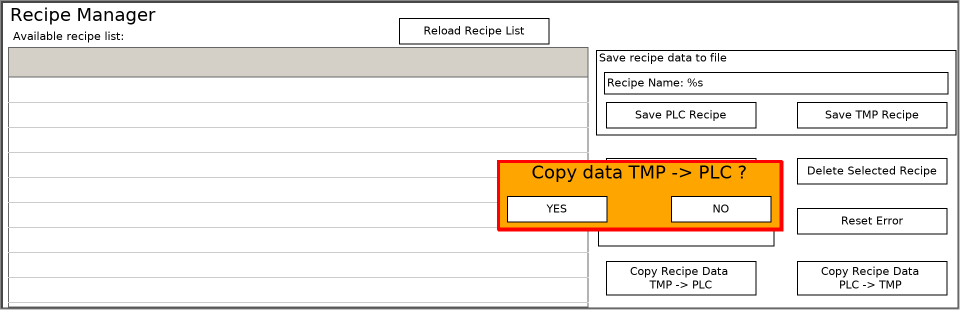
VISUALIZATION vRecManDialog_Wide  // 960x310
VAR_IN_OUT
	fbRecipe:fbRecMan;
END_VAR
    Rectangle (596,50 360x85), "Save recipe data to file"
    Table (8,47 580x260), data array: fbRecipe.astRecipeList
        p1128707560: fbRecipe.iNbOfFoundRecipes
        p1137915858: fbRecipe.iTableSelIndex
        p1822360349: fbRecipe.bTableRowSelected
        p3854506369: fbRecipe.astRecipeList[INDEX].sFileName
        p1892666644: fbRecipe.astRecipeList[INDEX].dtCreationTime
        p2232123230: Recipe Name
        p511219082: Creation Time
    Label (7,0 150x30), "Recipe Manager"
    Label (10,29 150x15), "Available recipe list:"
    RoundedRectangle (399,18 150x26), "Reload Recipe List", colour toggle: fbRecipe.bRefreshingRecipeList
        toggle fbRecipe.bReloadRecipes
    RoundedRectangle (606,102 150x26), "Save PLC Recipe", colour toggle: fbRecipe.bWritingRecipe
        OnMouseClick: execute { fbRecipe.bWriteRecipe := NOT fbRecipe.bWriteRecipe; fbRecipe.bSavePLCStruct := TRUE; }
    Rectangle (604,72 344x22), "Recipe Name: %s", text variable: fbRecipe.sRecipeName
        OnMouseClick: write fbRecipe.sRecipeName via Default, title 'New Recipe Name', format %s
    RoundedRectangle (606,261 150x34), "Copy Recipe Data TMP -> PLC", colour toggle: fbRecipe.bCopyTMP_2_PLC
        toggle fbRecipe.bCopyTMP_2_PLC
    RoundedRectangle (797,261 150x34), "Copy Recipe Data PLC -> TMP", colour toggle: fbRecipe.bCopyPLC_2_TMP
        toggle fbRecipe.bCopyPLC_2_TMP
    RoundedRectangle (606,158 150x26), "Read Selected Recipe", colour toggle: fbRecipe.bReadingRecipe
        toggle fbRecipe.bReadRecipe
    RoundedRectangle (797,102 150x26), "Save TMP Recipe", colour toggle: fbRecipe.bWritingRecipe
        OnMouseClick: execute { fbRecipe.bWriteRecipe := NOT fbRecipe.bWriteRecipe; fbRecipe.bSavePLCStruct := FALSE; }
    Rectangle (598,196 176x50), "Error: %s", text variable: fbRecipe.nErrorCode, invisible if: NOT fbRecipe.bError
        OnMouseClick: write fbRecipe.sRecipeName via Default, title 'New Recipe Name', format %s
    RoundedRectangle (797,208 150x26), "Reset Error", colour toggle: fbRecipe.bResetInternal, invisible if: NOT fbRecipe.bError
        toggle fbRecipe.bResetInternal
    RoundedRectangle (797,158 150x26), "Delete Selected Recipe", colour toggle: fbRecipe.bDeletingRecipe
        toggle fbRecipe.bDeleteRecipe
    Group (498,161 285x70), invisible if: NOT fbRecipe.bDeleteRecipe
        Rectangle (0,0 285x70), "Delete selection ?"
        RoundedRectangle (10,36 100x26), "YES"
            toggle fbRecipe.bDeleteConfirmed
        RoundedRectangle (174,36 100x26), "NO"
            toggle fbRecipe.bDeleteRecipe
    Rectangle (1,1 958x308)
    Group (497,160 285x70), invisible if: NOT fbRecipe.bCopyTMP_2_PLC
        Rectangle (0,0 285x70), "Copy data TMP -> PLC ?"
        RoundedRectangle (10,36 100x26), "YES"
            toggle fbRecipe.bCopyTMP_2_PLC_Confirmed
        RoundedRectangle (174,36 100x26), "NO"
            toggle fbRecipe.bCopyTMP_2_PLC
END_VISUALIZATION

(* stored: Version 1.1.0.1, ProductVersion 3.1.4024.12
   Visu vRecManDialog_Wide: Id {2e584d1c-6801-4b31-a55d-14a314c59b22} *)
